FUNCTION_BLOCK INTERNAL FINAL FB_RoundTripFloatTests EXTENDS FB_TestSuite
VAR CONSTANT
    cExpected : REAL := 13.37;
END_VAR
VAR
    fbWriteCtx      : FB_WriteContext;
    fbParseCtx      : FB_ParseContext;
    aBuffer         : ARRAY[0..15] OF BYTE;
    hrWriterActual  : HRESULT;
    hrParserActual  : HRESULT;
    fActual         : REAL;
END_VAR

TEST(__POUNAME());

// Arrange
fbWriteCtx.FromBuffer(aBuffer);
fbParseCtx.FromBuffer(aBuffer);
fbWriteCtx.refCtx.stState.nBufferPos := fbParseCtx.refCtx.stState.nBufferPos := 2;

// Act
hrWriterActual := F_WriteFloat(fbWriteCtx.refCtx.stBuffer, fbWriteCtx.refCtx.stState, cExpected);
hrParserActual := F_ParseFloat(fbParseCtx.refCtx, fVAlue=> fActual);

// Assert
AssertEquals_DINT(Expected:= S_OK, Actual:= hrWriterActual, Message:= 'Expected hrWriterActual = S_OK');
AssertEquals_DINT(Expected:= S_OK, Actual:= hrParserActual, Message:= 'Expected hrParserActual = S_OK');
AssertEquals_REAL(Expected:= cExpected, Actual:= fActual, Delta:= 1.0E-44, Message:= 'Values differ');

TEST_FINISHED_NAMED(__POUNAME());

END_FUNCTION_BLOCK

(* stored: Version 1.1.0.1
   POU FB_RoundTripFloatTests: Id {2c925fdb-d1b2-4454-938c-fb90f7c69610}, SpecialFunc None *)
